(* IEC 61131-3 sources: CodesysTest/alpha/export/FBs/Components/FunnelFB.pou/DelaySetting.prop, 1 file *)

(* ---- Set.pm.st ---- *)
(*#-#-#-#-#-#-#-#-#-#---Declaration---#-#-#-#-#-#-#-#-#-#-#-#-#*)

VAR
END_VAR
(*#-#-#-#-#-#-#-#-#-#---Implementation---#-#-#-#-#-#-#-#-#-#-#-#-#*)

openDelayTimer.PT := TO_TIME(DelaySetting * 1000);
